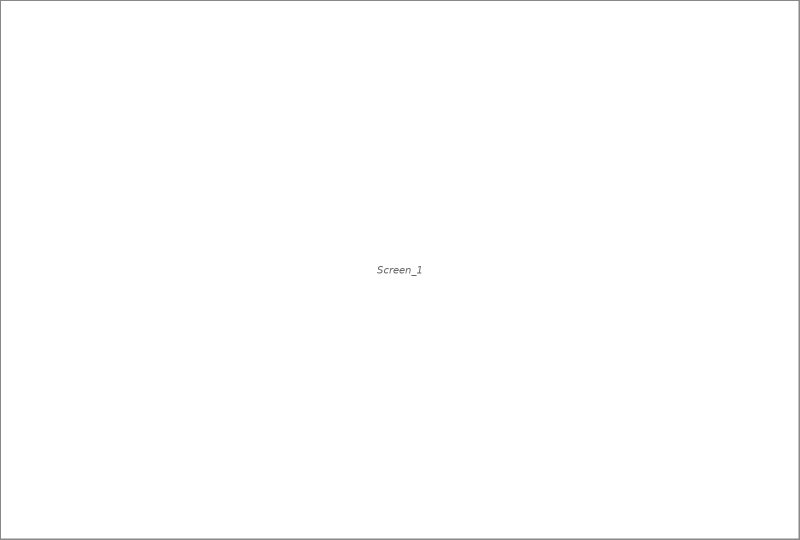
VISUALIZATION Screen_Maintenance  // 800x540
    TabControl (0,0 800x540), frame switch variable: GVL.HMI_Heading[1]
        shows Screen_1()
        shows Screen_2()
        shows Screen_3()
        [0]: TabTitle=Input Output
        [1]: TabTitle=Motor
        [2]: TabTitle=Diagram
END_VISUALIZATION

(* stored: Version 1.1.0.1, ProductVersion 3.1.4024.12
   Visu Screen_Maintenance: Id {ec18ebd9-cc0a-4d08-9916-28e5d740140e} *)
